// SIMATIC S7-200 project (STEP 7-Micro/WIN), CPU 224XP REL 02.01

SYMBOL_TABLE USUARIO1
PARO             I0.0
MARCHA           I0.1
LAMPARA_1        Q0.0
LAMPARA_2        Q0.1
LAMPARA_3        Q0.2
END_SYMBOL_TABLE

ORGANIZATION_BLOCK PRINCIPAL:OB1
TITLE=COMENTARIOS DEL PROGRAMA
BEGIN
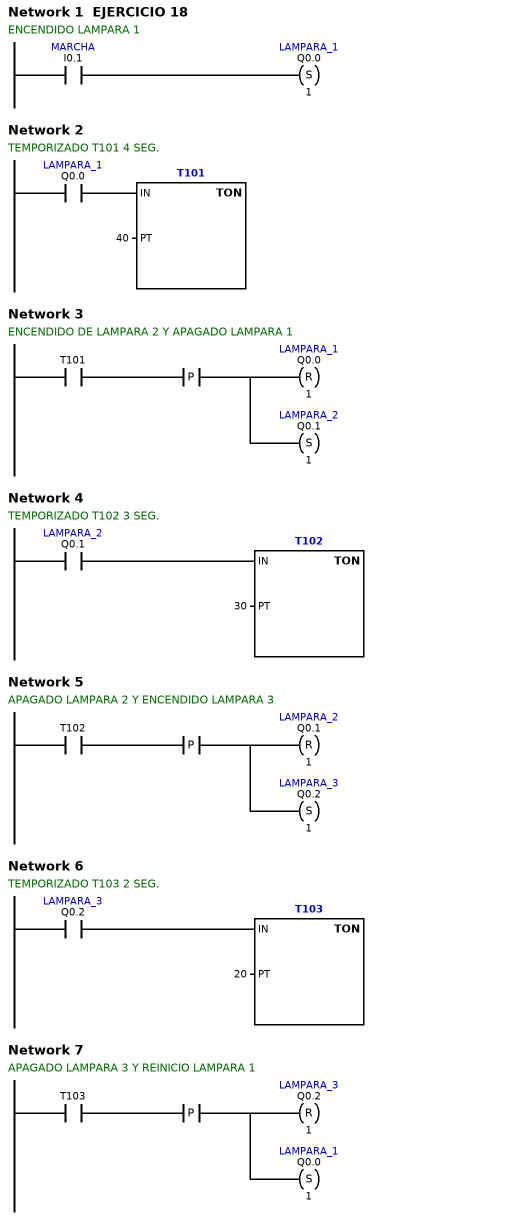
Network 1 // EJERCICIO 18
// ENCENDIDO LAMPARA 1
// (network saved uncompiled; LAD cells follow)
// row 0: c0 -| |- MARCHA:I0.1  c1 --  c2 -(S) LAMPARA_1:Q0.0, 1
Network 2
// TEMPORIZADO T101 4 SEG.
// (network saved uncompiled; LAD cells follow)
// row 0: c0 -| |- LAMPARA_1:Q0.0  c1 [TON T101 IN:=power@row0, PT:=40]
// row 1: c1 [box]
Network 3
//  ENCENDIDO DE LAMPARA 2 Y APAGADO LAMPARA 1
// (network saved uncompiled; LAD cells follow)
// row 0: c0 -| |- T101  c1 -|P|-  v  c2 -(R) LAMPARA_1:Q0.0, 1
// row 1: c1 ^  c2 -(S) LAMPARA_2:Q0.1, 1
Network 4
// TEMPORIZADO T102 3 SEG.
// (network saved uncompiled; LAD cells follow)
// row 0: c0 -| |- LAMPARA_2:Q0.1  c1 --  c2 [TON T102 IN:=power@row0, PT:=30]
// row 1: c2 [box]
Network 5
// APAGADO LAMPARA 2 Y ENCENDIDO LAMPARA 3 
// (network saved uncompiled; LAD cells follow)
// row 0: c0 -| |- T102  c1 -|P|-  v  c2 -(R) LAMPARA_2:Q0.1, 1
// row 1: c1 ^  c2 -(S) LAMPARA_3:Q0.2, 1
Network 6
// TEMPORIZADO T103 2 SEG.
// (network saved uncompiled; LAD cells follow)
// row 0: c0 -| |- LAMPARA_3:Q0.2  c1 --  c2 [TON T103 IN:=power@row0, PT:=20]
// row 1: c2 [box]
Network 7
// APAGADO LAMPARA 3 Y REINICIO LAMPARA 1
// (network saved uncompiled; LAD cells follow)
// row 0: c0 -| |- T103  c1 -|P|-  v  c2 -(R) LAMPARA_3:Q0.2, 1
// row 1: c1 ^  c2 -(S) LAMPARA_1:Q0.0, 1
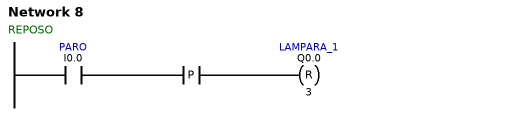
Network 8
// REPOSO
// (network saved uncompiled; LAD cells follow)
// row 0: c0 -| |- PARO:I0.0  c1 -|P|-  c2 -(R) LAMPARA_1:Q0.0, 3
END_ORGANIZATION_BLOCK
